FUNCTION_BLOCK iCreateDrive (* Service Interface Function Block Type *)
  (* Standard: 61499-2 *)
  (* Version 0.0, 2012-08-27, 4DIAC-IDE, 4DIAC-Consortium *)
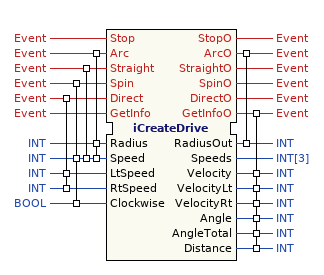
  EVENT_INPUT
    Stop;
    Arc WITH Speed, Radius; (* Drives in an arc. *)
    Straight WITH Speed; (* Drives straight at speed in mm/s *)
    Spin WITH Speed, Clockwise; (* spins Clockwise with edge speed of speed in mm/s according to Clockwise *)
    Direct WITH RtSpeed, LtSpeed; (* Drive each motoe/ wheel directiy *)
    GetInfo;
  END_EVENT
  EVENT_OUTPUT
    StopO;
    ArcO WITH RadiusOut;
    StraightO;
    SpinO;
    DirectO;
    GetInfoO WITH Velocity, VelocityLt, VelocityRt, Angle, AngleTotal, Distance;
  END_EVENT
  VAR_INPUT
    Radius : INT; (* Arc turning radius *)
    Speed : INT; (* speed (-500 to 500 mm/s) of both wheels *)
    LtSpeed : INT; (* Left Wheel speed (-500 to 500 mm/s) *)
    RtSpeed : INT; (* Right Wheel speed (-500 to 500 mm/s) *)
    Clockwise : BOOL; (* T=1=Clcokwise:; r *)
  END_VAR
  VAR_OUTPUT
    RadiusOut : INT; (* Turning radius used *)
    Speeds : ARRAY [0..2] OF INT; (* [both,Lt,Rt] wheel speeds *)
    Velocity : INT; (* wheel (both) velocity (speed) in mms *)
    VelocityLt : INT; (* Lt wheel velocity (speed) in mms *)
    VelocityRt : INT; (* Rt wheel velocity (speed) in mms *)
    Angle : INT; (* normalized angle *)
    AngleTotal : INT; (* accumulated angle *)
    Distance : INT; (* accumulated distance the Create has traveled since it was turned on *)
  END_VAR
  SERVICE APPLICATION/RESOURCE (* Service Interface Function Block Type *)
    SEQUENCE normal_establishment
      APPLICATION.INIT+(PARAMS) -> APPLICATION.INITO+(PARAMS);
    END_SEQUENCE
    SEQUENCE unsuccessful_establishment
      APPLICATION.INIT+(PARAMS) -> APPLICATION.INITO-(STATUS);
    END_SEQUENCE
    SEQUENCE request_confirm
      APPLICATION.REQ+(SD) -> APPLICATION.CNF+(RD);
    END_SEQUENCE
    SEQUENCE request_inhibited
      APPLICATION.REQ-(SD) -> APPLICATION.CNF-(STATUS);
    END_SEQUENCE
    SEQUENCE request_error
      APPLICATION.REQ+(SD) -> APPLICATION.CNF-(STATUS);
    END_SEQUENCE
    SEQUENCE indication_response
      RESOURCE.indicate(RD) -> APPLICATION.IND+(RD);
      APPLICATION.RSP(QI,SD) -> RESOURCE.response(QI,SD);
    END_SEQUENCE
    SEQUENCE indication_inhibited
      RESOURCE.indicate(RD,QI=FALSE) -> RESOURCE.inhibited();
    END_SEQUENCE
    SEQUENCE error_indication
      RESOURCE.error(STATUS) -> APPLICATION.IND-(STATUS);
    END_SEQUENCE
    SEQUENCE application_initiated_termination
      APPLICATION.INIT-() -> APPLICATION.INITO-(STATUS);
    END_SEQUENCE
    SEQUENCE resource_initiated_termination
      -> APPLICATION.INITO-(STATUS);
    END_SEQUENCE
  END_SERVICE
END_FUNCTION_BLOCK
